// Mitsubishi GX Works2 project: BookEX6_43 File   PLC: Q13UDV

// global labels: Global
VAR_GLOBAL
  bVar0 AT M5000 : BOOL;
  abArray0 AT M5010 : ARRAY [0..49] OF BOOL;
  sStr0 AT D5000 : STRING[199];
  sStr1 AT D5100 : STRING[199];
  sStr2 AT D5200 : STRING[199];
  sStr3 AT D5300 : STRING[199];
  sStr4 AT D5400 : STRING[199];
  sStr5 AT D5500 : STRING[199];
  sStr6 AT D5600 : STRING[199];
  sStr7 AT D5700 : STRING[199];
  sStr8 AT D5800 : STRING[199];
  sStr9 AT D5900 : STRING[199];
  iVar0 AT D4500 : INT;
  iVar1 AT D4501 : INT;
  iVar2 AT D4502 : INT;
  iVar3 AT D4503 : INT;
  iVar4 AT D4504 : INT;
  iVar5 AT D4505 : INT;
  iVar6 AT D4506 : INT;
  iVar7 AT D4507 : INT;
  iVar8 AT D4508 : INT;
  iVar9 AT D4509 : INT;
  dVar0 AT D4510 : DINT;
  dVar1 AT D4512 : DINT;
  dVar2 AT D4514 : DINT;
  dVar3 AT D4516 : DINT;
  dVar4 AT D4518 : DINT;
  dVar5 AT D4520 : DINT;
  dVar6 AT D4522 : DINT;
  dVar7 AT D4524 : DINT;
  dVar8 AT D4526 : DINT;
  dVar9 AT D4528 : DINT;
  wVar0 AT D4530 : WORD;
  wVar1 AT D4531 : WORD;
  wVar2 AT D4532 : WORD;
  wVar3 AT D4533 : WORD;
  wVar4 AT D4534 : WORD;
  wVar5 AT D4535 : WORD;
  wVar6 AT D4536 : WORD;
  wVar7 AT D4537 : WORD;
  wVar8 AT D4538 : WORD;
  wVar9 AT D4539 : WORD;
  dwVar0 AT D4540 : DWORD;
  dwVar1 AT D4542 : DWORD;
  dwVar2 AT D4544 : DWORD;
  dwVar3 AT D4546 : DWORD;
  dwVar4 AT D4548 : DWORD;
  dwVar5 AT D4550 : DWORD;
  dwVar6 AT D4552 : DWORD;
  dwVar7 AT D4554 : DWORD;
  dwVar8 AT D4556 : DWORD;
  dwVar9 AT D4558 : DWORD;
  fsVar0 AT D4560 : REAL;
  fsVar1 AT D4562 : REAL;
  fsVar2 AT D4564 : REAL;
  fsVar3 AT D4566 : REAL;
  fsVar4 AT D4568 : REAL;
  fsVar5 AT D4570 : REAL;
  fsVar6 AT D4572 : REAL;
  fsVar7 AT D4574 : REAL;
  fsVar8 AT D4576 : REAL;
  fsVar9 AT D4578 : REAL;
  fdVar0 AT D4580 : LREAL;
  tTime0 AT D4620 : TIME;
  tTime1 AT D4622 : TIME;
  tTime2 AT D4624 : TIME;
  tTime3 AT D4626 : TIME;
  tTime4 AT D4628 : TIME;
  tTime5 AT D4630 : TIME;
  tTime6 AT D4632 : TIME;
  tTime7 AT D4634 : TIME;
  tTime8 AT D4636 : TIME;
  tTime9 AT D4638 : TIME;
  tTime10 AT D4640 : TIME;
  bVar1 AT M5001 : BOOL;
  bVar2 AT M5002 : BOOL;
  bVar3 AT M5003 : BOOL;
  bVar4 AT M5004 : BOOL;
  bVar5 AT M5005 : BOOL;
  bVar6 AT M5006 : BOOL;
  bVar7 AT M5007 : BOOL;
  bVar8 AT M5008 : BOOL;
  bVar9 AT M5009 : BOOL;
  abArray1 AT M5060 : ARRAY [0..49] OF BOOL;
  abArray2 AT M5110 : ARRAY [0..49] OF BOOL;
  abArray3 AT M5160 : ARRAY [0..49] OF BOOL;
  abArray4 AT M5210 : ARRAY [0..49] OF BOOL;
  abArray5 AT M5260 : ARRAY [0..49] OF BOOL;
  abArray6 AT M5310 : ARRAY [0..49] OF BOOL;
  abArray7 AT M5360 : ARRAY [0..49] OF BOOL;
  abArray8 AT M5410 : ARRAY [0..49] OF BOOL;
  abArray9 AT M5460 : ARRAY [0..49] OF BOOL;
  fdVar1 AT D4584 : LREAL;
  fdVar2 AT D4588 : LREAL;
  fdVar3 AT D4592 : LREAL;
  fdVar4 AT D4596 : LREAL;
  fdVar5 AT D4600 : LREAL;
  fdVar6 AT D4604 : LREAL;
  fdVar7 AT D4608 : LREAL;
  fdVar8 AT D4612 : LREAL;
  fdVar9 AT D4616 : LREAL;
  afsPen0 AT D2000 : ARRAY [0..499] OF REAL;
  afsPen1 AT D3000 : ARRAY [0..499] OF REAL;
END_VAR

// task ExCDSET (event TRUE, interval 0, priority 31): ExQCDSET
// task ExQDRSET (event TRUE, interval 0, priority 31): ExQDRSET
// task ExRSET (event TRUE, interval 0, priority 31): ExRSET
// user libraries (not included): HMI

PROGRAM ExQCDSET
VAR
  Mov4INT_1 : Mov4INT;
END_VAR
(* structured ladder/FBD written out as ST: instructions are called as NAME(EN, inputs, outputs); _pN, _eN, _tN stand for wires *)
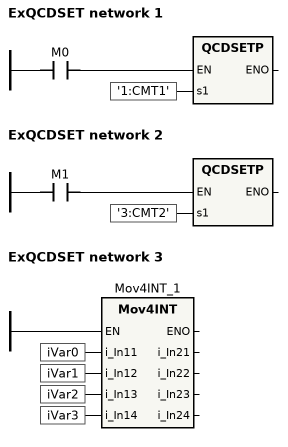
(* network 1 *)
QCDSETP(M0, '1:CMT1');
(* network 2 *)
QCDSETP(M1, '3:CMT2');
(* network 3 *)
Mov4INT_1(EN := TRUE, i_In11 := iVar0, i_In12 := iVar1, i_In13 := iVar2, i_In14 := iVar3);
END_PROGRAM

PROGRAM ExQDRSET
VAR
  Mov4WORD_1 : Mov4WORD;
  Mov4WORD_2 : Mov4WORD;
END_VAR
(* structured ladder/FBD written out as ST: instructions are called as NAME(EN, inputs, outputs); _pN, _eN, _tN stand for wires *)
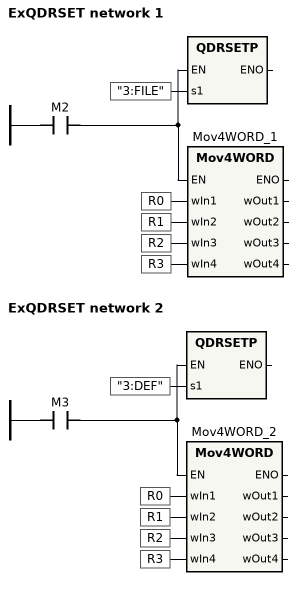
(* network 1 *)
QDRSETP(M2, "3:FILE");
Mov4WORD_1(EN := M2, wIn1 := R0, wIn2 := R1, wIn3 := R2, wIn4 := R3);
(* network 2 *)
QDRSETP(M3, "3:DEF");
Mov4WORD_2(EN := M3, wIn1 := R0, wIn2 := R1, wIn3 := R2, wIn4 := R3);
END_PROGRAM

PROGRAM ExRSET
VAR
  Mov4WORD_1 : Mov4WORD;
  Mov4WORD_2 : Mov4WORD;
  Mov4WORD_3 : Mov4WORD;
  Mov8WORD_1 : Mov8WORD;
END_VAR
(* structured ladder/FBD written out as ST: instructions are called as NAME(EN, inputs, outputs); _pN, _eN, _tN stand for wires *)
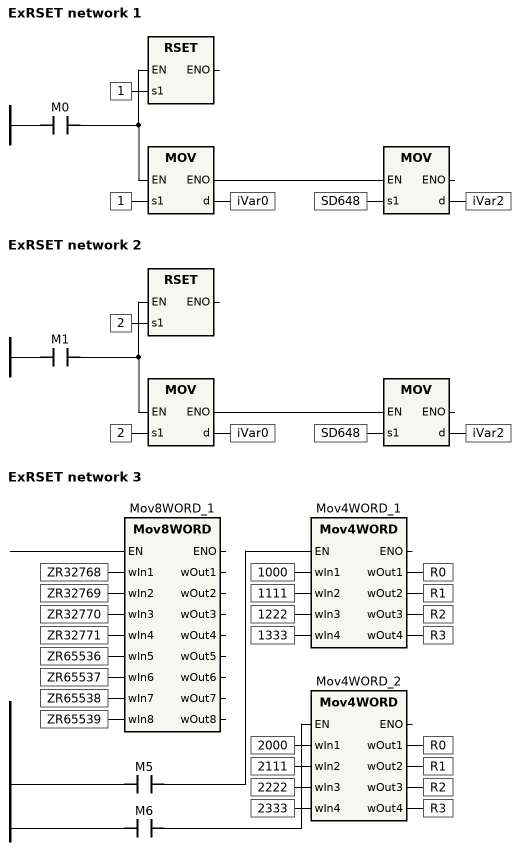
(* network 1 *)
RSET(M0, 1);
_e1 := MOV(M0, 1, iVar0);
MOV(_e1, SD648, iVar2);
(* network 2 *)
RSET(M1, 2);
_e1 := MOV(M1, 2, iVar0);
MOV(_e1, SD648, iVar2);
(* network 3 *)
Mov8WORD_1(EN := TRUE, wIn1 := ZR32768, wIn2 := ZR32769, wIn3 := ZR32770, wIn4 := ZR32771, wIn5 := ZR65536, wIn6 := ZR65537, wIn7 := ZR65538, wIn8 := ZR65539);
Mov4WORD_1(EN := M5, wIn1 := 1000, wIn2 := 1111, wIn3 := 1222, wIn4 := 1333, wOut1 => R0, wOut2 => R1, wOut3 => R2, wOut4 => R3);
Mov4WORD_2(EN := M6, wIn1 := 2000, wIn2 := 2111, wIn3 := 2222, wIn4 := 2333, wOut1 => R0, wOut2 => R1, wOut3 => R2, wOut4 => R3);
END_PROGRAM
